DEVICE_TYPE _TCREST
  (* Standard: 61499-2 *)
  (* Version 0.1, 2017-00-02, hpea485, UOA *)
  RESOURCE c : _Core
  END_RESOURCE
END_DEVICE_TYPE
